# EPICS substitutions: TPGSup/TPG300_channels.substitutions
file TPG300_channels.template {

pattern {PORT, P, CHAN, IFTEST, TPG_UNDERRANGE_ALARM_SEVERITY}
{"\$(PORT)", "\$(P)", "A1", "\$(IFPRESSURA1)", "\$(TPG_UNDERRANGE_ALARM_SEVERITY_CHAN1)"}
{"\$(PORT)", "\$(P)", "A2", "\$(IFPRESSURA2)", "\$(TPG_UNDERRANGE_ALARM_SEVERITY_CHAN2)"}
{"\$(PORT)", "\$(P)", "B1", "\$(IFPRESSURB1)", "\$(TPG_UNDERRANGE_ALARM_SEVERITY_CHAN1)"}
{"\$(PORT)", "\$(P)", "B2", "\$(IFPRESSURB2)", "\$(TPG_UNDERRANGE_ALARM_SEVERITY_CHAN2)"}
}
